Staubli VAL3: Binary7En.pjx

--- Binary7En.pjx ---
Parameters version=s7.7.2 stackSize=5000 millimeterUnit=true
Program file=BinToDec.pgx
Program file=BitWord.pgx
Program file=boolAnd.pgx
Program file=boolNand.pgx
Program file=boolNor.pgx
Program file=boolOr.pgx
Program file=boolXor.pgx
Program file=ChekCompBinary.pgx
Program file=DecToBin.pgx
Program file=DecToHex.pgx
Program file=DisplayResult.pgx
Program file=examplemenu.pgx
Program file=HexToDec.pgx
Program file=isBinary.pgx
Program file=isHexadecimal.pgx
Program file=pow.pgx
Program file=readme.pgx
Program file=RecFunction.pgx
Program file=shiftLeft.pgx
Program file=shiftRight.pgx
Program file=start.pgx
Program file=stop.pgx
Program file=SubMenu.pgx
Data file=Binary7En.dtx

--- Binary7En.dtx ---
bool bRead
public mdesc mNomSpeed
num nKey
string sBit[16] = "1010011010"
string sMenu[8]
  [2] = "F1: Decimal (num) to Binary (string)"
  [3] = "F2: Binary (string) to Decimal (num)"
  [4] = "F3: Operator function"
  [5] = "F4: Power calculation"
  [6] = "F5: And function (num and num)"
  [7] = "F6: Write 16 bit word"
string sSubMenu[7]
  [2] = "F1: And function"
  [3] = "F2: Or function"
  [4] = "F3: Xor function"
  [5] = "F4: Nand function"
  [6] = "F5: Nor function"
string sDec2HexSymbols[16]
  [0] = "0"
  [1] = "1"
  [2] = "2"
  [3] = "3"
  [4] = "4"
  [5] = "5"
  [6] = "6"
  [7] = "7"
  [8] = "8"
  [9] = "9"
  [10] = "A"
  [11] = "B"
  [12] = "C"
  [13] = "D"
  [14] = "E"
  [15] = "F"
string sDecHexBuff
string sHexDecBuff
num nHex2DecSymbols{}
  [0] = {}
  [1] = 1
  [8] = 8
  [9] = 9
  [A] = 10
  [B] = 11
  [C] = 12
  [D] = 13
  [E] = 14
  [F] = 15
  [2] = 2
  [3] = 3
  [4] = 4
  [5] = 5
  [6] = 6
  [7] = 7

--- BitWord.pgx ---
public program BitWord(num x_nDecimal, string& x_sBinary[])
  local num l_ni
  local string l_sVal
begin
  //-----------------------------------------------------------------------
  //Header begin
  //Description of program
  //  This program turns a decimal number into a binary word.
  //  Receives decimal value and turns it into the corresponding
  //  binary word (16 Bits).
  //
  //Input parameters
  //  num x_nDecimal :
  //    role : decimal value to convert
  //
  //Output parameters
  //  string x_sBinary :
  //    role : binary value converted (16 Bits)
  //
  //Example
  //  BitWord(78,sBinaryValue)
  //
  //History
  //  Creation : 16-04-09 - t.Gra
  //Header end
  //-----------------------------------------------------------------------
  //take the full value
  x_nDecimal=roundDown(x_nDecimal)
  //Calcul loop
  do
    if (x_nDecimal%2)==0
      x_sBinary="0"+x_sBinary
    else
      x_sBinary="1"+x_sBinary
    endIf
    x_nDecimal=roundDown(x_nDecimal/2)
  until (x_nDecimal<1)
  l_sVal=x_sBinary
  //Add bit 0
  for l_ni=1 to (16-len(l_sVal))
    x_sBinary="0"+x_sBinary
  endFor
end

--- boolNand.pgx ---
public program boolNand(string x_sBinary1, string x_sBinary2, string& x_sReturn[])
  local num l_nNumBit
  local string l_sValsup
  local string l_sValmin
begin
  //-----------------------------------------------------------------------
  //Header begin
  //Description of program
  //  This program provides a Nand logical operator for 2 binary values.
  //
  //     0 and 0 = 1
  //     0 and 1 = 1
  //     1 and 1 = 0
  //
  //Input parameters
  //  string x_sBinary1 :
  //    role : 1 st binary number
  //  string x_sBinary2 :
  //    role : 2 nd binary number
  //
  //Output parameters
  //  string x_sReturn :
  //    role : Result of calculation x_sBinary1 NAND x_sBinary2
  //
  //Example
  //  Nand("10101011","00011011",sResult)
  //
  //History
  //  Creation : 16-04-09 - t.Gra
  //Header end
  //-----------------------------------------------------------------------
  //Initialization
  l_nNumBit=0
  l_sValsup=""
  l_sValmin=""
  x_sReturn=""
  //call function for error control
  call ChekCompBinary(x_sBinary1,x_sBinary2,l_sValsup,l_sValmin)
  //calcul loop
  if (bRead==true)
    for l_nNumBit=(len(l_sValsup)-1) to 0 step -1
      if ((mid(l_sValsup,1,l_nNumBit)=="1") and (mid(l_sValmin,1,l_nNumBit)=="1"))
        x_sReturn="0"+x_sReturn
      else
        x_sReturn="1"+x_sReturn
      endIf
    endFor
  else
    x_sReturn="Error"
  endIf
end

--- boolOr.pgx ---
public program boolOr(string x_sBinary1, string x_sBinary2, string& x_sReturn[])
  local num l_nNumBit
  local string l_sValsup
  local string l_sValmin
begin
  //-----------------------------------------------------------------------
  //Header begin
  //Description of program
  //  This program provides an Or logical operator for 2 binary values.
  //
  //     0 or 0 = 0
  //     0 or 1 = 1
  //     1 or 1 = 1
  //
  //Input parameters
  //  string x_sBinary1 :
  //    role : 1 st binary number
  //  string x_sBinary2 :
  //    role : 2 nd binary number
  //
  //Output parameters
  //  string x_sReturn :
  //    role : Result of calculation x_sBinary1 OR x_sBinary2
  //
  //Example
  //  Or("10101011","00011011",sResult)
  //
  //History
  //  Creation : 16-04-09 - t.Gra
  //Header end
  //-----------------------------------------------------------------------
  //Initialization
  l_nNumBit=0
  l_sValsup=""
  l_sValmin=""
  //call function for error control
  call ChekCompBinary(x_sBinary1,x_sBinary2,l_sValsup,l_sValmin)
  //calcul loop
  if (bRead==true)
    for l_nNumBit=(len(l_sValsup)-1) to 0 step -1
      if ((mid(l_sValsup,1,l_nNumBit)=="0") and (mid(l_sValmin,1,l_nNumBit)=="0"))
        x_sReturn="0"+x_sReturn
      else
        x_sReturn="1"+x_sReturn
      endIf
    endFor
  else
    x_sReturn="Error"
  endIf
end

--- DecToBin.pgx ---
public program DecToBin(num x_nDecimal, string& x_sBinary[])
begin
  //-----------------------------------------------------------------------
  //Header begin
  //Description of program
  //  This program turns a decimal number into a binary word.
  //  Receives decimal value and turns it into the corresponding
  //  binary word.
  //
  //Input parameters
  //  num x_nDecimal :
  //    role : decimal value to convert
  //
  //Output parameters
  //  string x_sBinary :
  //    role : binary value converted
  //
  //Example
  //  DecToBin(42,sBinaryValue)
  //
  //History
  //  Creation : 16-04-09 - t.Gra
  //Header end
  //-----------------------------------------------------------------------
  //take the full value
  x_nDecimal=roundDown(x_nDecimal)
  //Calcul loop
  do
    if (x_nDecimal%2)==0
      x_sBinary="0"+x_sBinary
    else
      x_sBinary="1"+x_sBinary
    endIf
    x_nDecimal=roundDown(x_nDecimal/2)
  until (x_nDecimal<1)
end

--- DecToHex.pgx ---
public program DecToHex(num x_nDecimal, string& x_sHex)
  local num l_nRest
  local num l_nDecimal
  local num l_nIndex
begin

  //only integers allowed!
  l_nDecimal = round(x_nDecimal)
  resize(sDecHexBuff, 1, 1)

  while l_nDecimal != 0

    l_nRest = l_nDecimal % 16
    sDecHexBuff[size(sDecHexBuff)-1] = sDec2HexSymbols[l_nRest]
    append(sDecHexBuff)
    l_nDecimal = roundDown(l_nDecimal/16)

  endWhile

  x_sHex = ""
  for l_nIndex = size(sDecHexBuff)-1 to 0 step-1
    x_sHex = x_sHex + sDecHexBuff[l_nIndex]
  endFor


end

--- HexToDec.pgx ---
public program HexToDec(string x_sHex, num& x_nDecimal)
  local num l_nIndex
  local num l_nResult
  local bool l_bIsHex
begin

  //upgrade: trim the input string!

  l_bIsHex=false
  call isHexadecimal(x_sHex, l_bIsHex)

  if l_bIsHex
    for l_nIndex=len(x_sHex)-1 to 0 step-1
      l_nResult = l_nResult + (nHex2DecSymbols[mid(x_sHex, 1, l_nIndex)]*power(16, len(x_sHex)-l_nIndex-1))
    endFor
    x_nDecimal = l_nResult
  else
    logMsg("Binary->HexToDec: wrong input format")
  endIf

end

--- isBinary.pgx ---
program isBinary(string x_sBinary, bool& x_bRes)
  local num l_nIndex
begin

  for l_nIndex= 0 to len(x_sBinary)-1
    if mid(x_sBinary, 1, l_nIndex)!="0" and mid(x_sBinary, 1, l_nIndex)!="1"
      x_bRes = false
      return
    endIf
  endFor

  x_bRes = true

end

--- readme.pgx ---
program readme()
begin
  //Title: Mathematical and Binary functions
  //
  //General description :
  //  This library provides a functions for binary and mathematical
  //  calculations.
  //
  //  1) transforms a binary to a decimal or vice-versa
  //  2) provides OR, XOR, AND operators for binary calculation
  //  3) Exponent Calculation
  //
  //Hardware required :
  //  - Robot system    : no specific robot system
  //  - Peripherals     : no peripherals required
  //
  //VAL3 options :
  //  - VAL3 version    : 7.*
  //  - VAL3 licenses   : no licenses required
  //  - VAL3 add-ons    : none
  //
  //Library version     : 7.6.1.0
  //
  //Public variables    : none
  //
  //Included libraries  : none
  //
  //Miscellaneous       : ---
  //
  //Keywords            : calculation, Operator, And, Or, Xor, Decimal, binary,
  //                      function, word.
end

--- shiftLeft.pgx ---
public program shiftLeft(string& x_sBinary, num x_nPos)
  local bool l_bIsBinary
  local string l_sBinary
  local num l_nIndex
begin

  l_bIsBinary=false
  call isBinary(x_sBinary, l_bIsBinary)
  l_sBinary = x_sBinary

  if l_bIsBinary
    for l_nIndex=0 to x_nPos-1
      l_sBinary = l_sBinary + "0"
    endFor
    x_sBinary=right(l_sBinary, len(x_sBinary))
  else
    logMsg("Binary->shiftLeft: wrong input format")
  endIf

end

--- shiftRight.pgx ---
public program shiftRight(string& x_sBinary, num x_nPos)
  local bool l_bIsBinary
  local string l_sBinary
  local num l_nIndex
begin

  l_bIsBinary=false
  call isBinary(x_sBinary, l_bIsBinary)
  l_sBinary = x_sBinary

  if l_bIsBinary
    for l_nIndex=0 to x_nPos-1
      l_sBinary = "0"+l_sBinary
    endFor
    x_sBinary=left(l_sBinary, len(x_sBinary))
  else
    logMsg("Binary->shiftLeft: wrong input format")
  endIf

end
